// TwinCAT 3 PLC project GOV_DAQ
// ProgramVersion: 3.1.4024.0
// libraries:
//   Tc2_Coupler, * (Beckhoff Automation GmbH)
//   Tc2_SPA, * (Beckhoff Automation GmbH)
//   Tc2_Standard, * (Beckhoff Automation GmbH)
//   Tc2_System, * (Beckhoff Automation GmbH)
//   Tc2_Utilities, * (Beckhoff Automation GmbH)
//   Tc3_Module, * (Beckhoff Automation GmbH)
// project tree:
//   GVLs/ GVL.TcGVL
//   / PlcTask.TcTTO
//   POUs/ MAIN.TcPOU
// real-time tasks:
//   TASK PlcTask: cycle T#10ms, priority 20, ADS port 350
//   TASK PlcTask1: cycle T#10ms, priority 21, ADS port 351
// I/O:
//   DEVICE Device 1 (EtherCAT), AmsNetId 5.141.19.14.2.1
//     Term 1 (EK1200) [EK1200-5000 EtherCAT Power supply (2A E-Bus)]
//       Term 2 (EL1809) [EL1809 16Ch. Dig. Input 24V, 3ms]
//       Term 3 (EL3114) [EL3114 4Ch. Ana. Input 0-20mA Diff.]
//       Term 4 (EL3104) [EL3104 4Ch. Ana. Input +/-10V Diff.]
//       Term 5 (EL9011) [EL9011 End Terminal]
// variable links:
//   GOV_DAQ/GOV_DAQ Instance <-> Device 1 (EtherCAT)/Term 1 (EK1200)/Term 3 (EL3114)
//     PlcTask Inputs/GVL.nCurrent_Input1 <-> AI Standard Channel 1/Value
//   GOV_DAQ/GOV_DAQ Instance <-> Device 1 (EtherCAT)/Term 1 (EK1200)/Term 4 (EL3104)
//     PlcTask Inputs/GVL.nVoltage_Input1 <-> AI Standard Channel 1/Value
//     PlcTask Inputs/GVL.nVoltage_Input2 <-> AI Standard Channel 2/Value

CONFIGURATION GOV_DAQ
    RESOURCE PLC ON TwinCAT3
        TASK PlcTask(INTERVAL := T#10ms, PRIORITY := 21);
        PROGRAM MAIN WITH PlcTask : MAIN;
    END_RESOURCE
END_CONFIGURATION

// ---- GVLs/GVL.TcGVL
{attribute 'qualified_only'}
VAR_GLOBAL
	
(* Digital Input variables for EL1809 *)
bDigital_Input1 AT %I* : BOOL;
bDigital_Input2 AT %I* : BOOL;
bDigital_Input3 AT %I* : BOOL;
bDigital_Input4 AT %I* : BOOL;
bDigital_Input5 AT %I* : BOOL;
bDigital_Input6 AT %I* : BOOL;
bDigital_Input7 AT %I* : BOOL;
bDigital_Input8 AT %I* : BOOL;
bDigital_Input9 AT %I* : BOOL;
bDigital_Input10 AT %I* : BOOL;
bDigital_Input11 AT %I* : BOOL;
bDigital_Input12 AT %I* : BOOL;
bDigital_Input13 AT %I* : BOOL;
bDigital_Input14 AT %I* : BOOL;
bDigital_Input15 AT %I* : BOOL;
bDigital_Input16 AT %I* : BOOL;

(*4-20 mA Analog inputs for EL3114*)
nCurrent_Input1 AT %I* : INT;
nCurrent_Input2 AT %I* : INT;
nCurrent_Input3 AT %I* : INT;
nCurrent_Input4 AT %I* : INT;

//Converted from DAQ resolution to engineering unit (mA)
rCurrent_Input1_EU AT %I* : REAL;
rCurrent_Input2_EU AT %I* : REAL;
rCurrent_Input3_EU AT %I* : REAL;
rCurrent_Input4_EU AT %I* : REAL;

(*0-10V Analog Input for EL3104*)
nVoltage_Input1 AT %I* : INT;
nVoltage_Input2 AT %I* : INT;
nVoltage_Input3 AT %I* : INT;
nVoltage_Input4 AT %I* : INT;

//Converted from DAQ resolution to engineering unit (V)
rVoltage_Input1_EU AT %I* : REAL;
rVoltage_Input2_EU AT %I* : REAL;
rVoltage_Input3_EU AT %I* : REAL;
rVoltage_Input4_EU AT %I* : REAL;

END_VAR

// ---- POUs/MAIN.TcPOU
(*
Purpose: (1) Takes 4-20mA as an input AND scales TO output a %Position assuming a linear relationship
		 (2) 

Inputs: (1) Servo-motor position indicator 4-20mA innput to EL3114
		(2) .... (0-10 V) input to EL3104

Outputs: No physical outputs. DAQ acquires data, processes it, and displays it as scope data. 
		 Users can may optionally use analytics tooling available in TwinCAT 3. Otherwise, data
		 can be exported as a .CSV file for analysis/record purposes in programs such as Excel or
		 MATLAB.

Notes:
(1) There is some fixed error in the calculation - 100% is never reach, but we get close ~99.9%!
(2) There are overcurrent protections (fuses) but no external overvoltage protections. Please double check
	the EL3104 will not be damaged with max input voltage of proccess variable being measured (card 
	can handle max. 10V)

*)

PROGRAM MAIN
VAR CONSTANT
	startVal_mA : REAL := 6350;
	rDAQtomA : REAL := (20 - 4)/(32768.0 - startVal_mA);
END_VAR


VAR
	
END_VAR

END_PROGRAM
